TYPE TupleStruct1:
    STRUCT
        field1: TupleStruct;
        field2: REAL;
    END_STRUCT;
END_TYPE
